	W =    -2.744 deg,	P =    30.268 deg,	R =  -167.022 deg
   GP2:
	UF : 1, UT : 1,
	J1=    90.000 deg,	J2=   -90.000 deg
};
P[599]{
   GP1:
	UF : 1, UT : 1,		CONFIG : 'N U T, 0, 0, 0',
	X =  2391.109  mm,	Y =   106.727  mm,	Z =   -21.577  mm,
	W =   -47.008 deg,	P =     6.653 deg,	R =   -83.994 deg
   GP2:
	UF : 1, UT : 1,
	J1=    83.000 deg,	J2=   -90.000 deg
};
P[600]{
   GP1:
	UF : 1, UT : 1,		CONFIG : 'N U T, 0, 0, 0',
	X =  2390.648  mm,	Y =   140.871  mm,	Z =   -20.910  mm,
	W =   -47.989 deg,	P =     7.881 deg,	R =   -87.078 deg
   GP2:
	UF : 1, UT : 1,
	J1=    83.000 deg,	J2=   -90.000 deg
};
P[601]{
   GP1:
	UF : 1, UT : 1,		CONFIG : 'N U T, 0, 0, 0',
	X =  2393.525  mm,	Y =   163.570  mm,	Z =   -20.785  mm,
	W =   -47.988 deg,	P =     7.880 deg,	R =  -106.126 deg
   GP2:
	UF : 1, UT : 1,
	J1=    83.000 deg,	J2=   -90.000 deg
};
P[602]{
   GP1:
	UF : 1, UT : 1,		CONFIG : 'N U T, 0, 0, 0',
	X =  2366.142  mm,	Y =   180.100  mm,	Z =    -9.199  mm,
	W =   -44.813 deg,	P =    -4.559 deg,	R =    -2.484 deg
   GP2:
	UF : 1, UT : 1,
	J1=    90.000 deg,	J2=   -90.000 deg
};
P[603]{
   GP1:
	UF : 1, UT : 1,		CONFIG : 'N U T, 0, 0, 0',
	X =  2505.035  mm,	Y =   180.287  mm,	Z =    -9.109  mm,
	W =   -44.818 deg,	P =    -4.562 deg,	R =    -2.490 deg
   GP2:
	UF : 1, UT : 1,
	J1=    90.000 deg,	J2=   -90.000 deg
};
P[604]{
   GP1:
	UF : 1, UT : 1,		CONFIG : 'N U T, 0, 0, 0',
	X =  2363.074  mm,	Y =    82.607  mm,	Z =    -8.621  mm,
	W =   -44.379 deg,	P =     8.160 deg,	R =    14.035 deg
   GP2:
	UF : 1, UT : 1,
	J1=    90.000 deg,	J2=   -90.000 deg
};
P[605]{
   GP1:
	UF : 1, UT : 1,		CONFIG : 'N U T, 0, 0, 0',
	X =  2414.311  mm,	Y =    81.629  mm,	Z =    -8.521  mm,
	W =   -44.393 deg,	P =     8.163 deg,	R =    14.043 deg
   GP2:
	UF : 1, UT : 1,
	J1=    90.000 deg,	J2=   -90.000 deg
};
P[606]{
   GP1:
	UF : 1, UT : 1,		CONFIG : 'N U T, 0, 0, 0',
	X =  2420.856  mm,	Y =    84.559  mm,	Z =    -6.348  mm,
	W =   -44.535 deg,	P =    -7.128 deg,	R =    33.228 deg
   GP2:
	UF : 1, UT : 1,
	J1=    90.000 deg,	J2=   -90.000 deg
};
P[607]{
   GP1:
	UF : 1, UT : 1,		CONFIG : 'N U T, 0, 0, 0',
	X =  2096.605  mm,	Y =  -181.583  mm,	Z =   897.867  mm,
	W =     -.064 deg,	P =    31.734 deg,	R =  -164.129 deg
   GP2:
	UF : 1, UT : 1,
	J1=    90.000 deg,	J2=   -90.000 deg
};
P[608]{
   GP1:
	UF : 1, UT : 1,		CONFIG : 'N U T, 0, 0, 0',
	X =  2114.149  mm,	Y =  -253.336  mm,	Z =   921.197  mm,
	W =     1.157 deg,	P =    35.359 deg,	R =   -90.786 deg
   GP2:
	UF : 1, UT : 1,
	J1=    90.000 deg,	J2=   -90.000 deg
};
P[609]{
   GP1:
	UF : 1, UT : 1,		CONFIG : 'N U T, 0, 0, 0',
	X =  2347.090  mm,	Y =    54.696  mm,	Z =   840.157  mm,
	W =    45.388 deg,	P =    17.262 deg,	R =    -1.525 deg
   GP2:
	UF : 1, UT : 1,
	J1=    90.000 deg,	J2=   -90.000 deg
};
P[610]{
   GP1:
	UF : 1, UT : 1,		CONFIG : 'N U T, 0, 0, 0',
	X =  2407.727  mm,	Y =    84.771  mm,	Z =   840.157  mm,
	W =    45.388 deg,	P =    17.262 deg,	R =    -1.525 deg
   GP2:
	UF : 1, UT : 1,
	J1=    90.000 deg,	J2=   -90.000 deg
};
P[611]{
   GP1:
	UF : 1, UT : 1,		CONFIG : 'N U T, 0, 0, 0',
	X =  2411.910  mm,	Y =    90.376  mm,	Z =   839.563  mm,
	W =     1.454 deg,	P =    40.369 deg,	R =    26.792 deg
   GP2:
	UF : 1, UT : 1,
	J1=    90.000 deg,	J2=   -90.000 deg
};
P[612]{
   GP1:
	UF : 1, UT : 1,		CONFIG : 'N U T, 0, 0, 0',
	X =  2400.458  mm,	Y =   114.292  mm,	Z =   839.623  mm,
	W =     1.448 deg,	P =    40.366 deg,	R =    26.776 deg
   GP2:
	UF : 1, UT : 1,
	J1=    90.000 deg,	J2=   -90.000 deg
};
P[613]{
   GP1:
	UF : 1, UT : 1,		CONFIG : 'N U T, 0, 0, 0',
	X =  2330.795  mm,	Y =    79.737  mm,	Z =   841.199  mm,
	W =   -50.335 deg,	P =   -10.786 deg,	R =    47.268 deg
   GP2:
	UF : 1, UT : 1,
	J1=    90.000 deg,	J2=   -90.000 deg
};
P[614]{
   GP1:
	UF : 1, UT : 1,		CONFIG : 'N U T, 0, 0, 0',
	X =  2394.366  mm,	Y =   112.525  mm,	Z =   840.958  mm,
	W =   -50.044 deg,	P =   -12.807 deg,	R =    45.682 deg
   GP2:
	UF : 1, UT : 1,
	J1=    90.000 deg,	J2=   -90.000 deg
};
P[615]{
   GP1:
	UF : 1, UT : 1,		CONFIG : 'N U T, 0, 0, 0',
	X =  2010.656  mm,	Y =   -98.489  mm,	Z =    -6.723  mm,
	W =    40.376 deg,	P =    23.931 deg,	R =    74.346 deg
   GP2:
	UF : 1, UT : 1,
	J1=    90.000 deg,	J2=  -100.000 deg
};
P[616]{
   GP1:
	UF : 1, UT : 1,		CONFIG : 'N U T, 0, 0, 0',
	X =  2009.129  mm,	Y =   124.302  mm,	Z =   -44.627  mm,
	W =    45.687 deg,	P =     4.511 deg,	R =    78.829 deg
   GP2:
	UF : 1, UT : 1,
	J1=    90.000 deg,	J2=  -100.000 deg
};
P[617]{
   GP1:
	UF : 1, UT : 1,		CONFIG : 'N U T, 0, 0, 0',
	X =  2230.271  mm,	Y =   -64.539  mm,	Z =    -1.822  mm,
	W =    44.892 deg,	P =    -3.427 deg,	R =     3.436 deg
   GP2:
	UF : 1, UT : 1,
	J1=    90.000 deg,	J2=   -90.000 deg
};
P[618]{
   GP1:
	UF : 1, UT : 1,		CONFIG : 'N U T, 0, 0, 0',
	X =  2628.655  mm,	Y =   126.905  mm,	Z =   907.127  mm,
	W =    31.997 deg,	P =    23.849 deg,	R =   -38.788 deg
   GP2:
	UF : 1, UT : 1,
	J1=    90.000 deg,	J2=   -90.000 deg
};
P[619]{
   GP1:
	UF : 1, UT : 1,		CONFIG : 'N U T, 0, 0, 0',
	X =   949.417  mm,	Y =    74.708  mm,	Z =  1003.698  mm,
	W =    14.657 deg,	P =    21.488 deg,	R =   -36.321 deg
   GP2:
	UF : 1, UT : 1,
	J1=    90.000 deg,	J2=   -90.000 deg
};
P[620]{
   GP1:
	UF : 1, UT : 1,		CONFIG : 'N U T, 0, 0, 0',
	X =   931.440  mm,	Y =   198.476  mm,	Z =   335.127  mm,
	W =   -34.527 deg,	P =    19.136 deg,	R =    25.896 deg
   GP2:
	UF : 1, UT : 1,
	J1=    90.000 deg,	J2=   -90.000 deg
};
P[621]{
   GP1:
	UF : 1, UT : 1,		CONFIG : 'N U T, 0, 0, 0',
	X =  1700.688  mm,	Y =   121.333  mm,	Z =   177.127  mm,
	W =   -48.737 deg,	P =     8.784 deg,	R =     7.978 deg
   GP2:
	UF : 1, UT : 1,
	J1=    90.000 deg,	J2=   -90.000 deg
};
P[622]{
   GP1:
	UF : 1, UT : 1,		CONFIG : 'N U T, 0, 0, 0',
	X =  2260.320  mm,	Y =   -63.687  mm,	Z =    -1.783  mm,
	W =    44.897 deg,	P =    -3.424 deg,	R =     3.430 deg
   GP2:
	UF : 1, UT : 1,
	J1=    90.000 deg,	J2=   -90.000 deg
};
P[623]{
   GP1:
	UF : 1, UT : 1,		CONFIG : 'N U T, 0, 0, 0',
	X =  2134.875  mm,	Y =   -62.293  mm,	Z =   -12.089  mm,
	W =    44.886 deg,	P =     3.630 deg,	R =    -4.912 deg
   GP2:
	UF : 1, UT : 1,
	J1=    90.000 deg,	J2=   -90.000 deg
};
P[624]{
   GP1:
	UF : 1, UT : 1,		CONFIG : 'N U T, 0, 0, 0',
	X =  2205.171  mm,	Y =   -64.816  mm,	Z =   -10.170  mm,
	W =    44.886 deg,	P =     3.630 deg,	R =    -4.912 deg
   GP2:
	UF : 1, UT : 1,
	J1=    90.000 deg,	J2=   -90.000 deg
};
P[625]{
   GP1:
	UF : 1, UT : 1,		CONFIG : 'N U T, 0, 0, 0',
	X =  2212.120  mm,	Y =   -62.897  mm,	Z =   -10.890  mm,
	W =    44.886 deg,	P =     3.630 deg,	R =   -11.550 deg
   GP2:
	UF : 1, UT : 1,
	J1=    90.000 deg,	J2=   -90.000 deg
};
P[626]{
   GP1:
	UF : 1, UT : 1,		CONFIG : 'N U T, 0, 0, 0',
	X =  1922.982  mm,	Y =    80.524  mm,	Z =   163.198  mm,
	W =   -51.903 deg,	P =     9.364 deg,	R =    21.482 deg
   GP2:
	UF : 1, UT : 1,
	J1=    90.000 deg,	J2=   -90.000 deg
};
P[627]{
   GP1:
	UF : 1, UT : 1,		CONFIG : 'N U T, 0, 0, 0',
	X =  2179.982  mm,	Y =    80.524  mm,	Z =   163.199  mm,
	W =   -51.227 deg,	P =   -13.564 deg,	R =     3.543 deg
   GP2:
	UF : 1, UT : 1,
	J1=    90.000 deg,	J2=   -90.000 deg
};
P[628]{
   GP1:
	UF : 1, UT : 1,		CONFIG : 'N U T, 0, 0, 0',
	X =  1984.534  mm,	Y =   -65.727  mm,	Z =   -17.955  mm,
	W =    44.885 deg,	P =     3.628 deg,	R =    -8.844 deg
   GP2:
	UF : 1, UT : 1,
	J1=    90.000 deg,	J2=   -90.000 deg
};
P[629]{
   GP1:
	UF : 1, UT : 1,		CONFIG : 'N U T, 0, 0, 0',
	X =  2097.268  mm,	Y =   -65.065  mm,	Z =   -17.473  mm,
	W =    44.885 deg,	P =     3.628 deg,	R =    -8.844 deg
   GP2:
	UF : 1, UT : 1,
	J1=    90.000 deg,	J2=   -90.000 deg
};
P[630]{
   GP1:
	UF : 1, UT : 1,		CONFIG : 'N U T, 0, 0, 0',
	X =  2179.963  mm,	Y =     8.530  mm,	Z =    59.476  mm,
	W =   -44.735 deg,	P =    -5.491 deg,	R =    -5.516 deg
   GP2:
	UF : 1, UT : 1,
	J1=    90.000 deg,	J2=   -90.000 deg
};
P[631]{
   GP1:
	UF : 1, UT : 1,		CONFIG : 'N U T, 0, 0, 0',
	X =  2112.828  mm,	Y =   -64.584  mm,	Z =   -16.753  mm,
	W =    41.205 deg,	P =   -19.972 deg,	R =    -8.013 deg
   GP2:
	UF : 1, UT : 1,
	J1=    90.000 deg,	J2=   -90.000 deg
};
P[632]{
   GP1:
	UF : 1, UT : 1,		CONFIG : 'N U T, 0, 0, 0',
	X =  2071.831  mm,	Y =  -111.826  mm,	Z =   -18.286  mm,
	W =   -37.503 deg,	P =      .971 deg,	R =    76.661 deg
   GP2:
	UF : 1, UT : 1,
	J1=    90.000 deg,	J2=   -90.000 deg
};
P[633]{
   GP1:
	UF : 1, UT : 1,		CONFIG : 'N U T, 0, 0, 0',
	X =  2101.801  mm,	Y =   -84.456  mm,	Z =   -18.286  mm,
	W =   -37.503 deg,	P =      .971 deg,	R =    85.242 deg
   GP2:
	UF : 1, UT : 1,
	J1=    90.000 deg,	J2=   -90.000 deg
};
P[634]{
   GP1:
	UF : 1, UT : 1,		CONFIG : 'N U T, 0, 0, 0',
	X =  2083.048  mm,	Y =     5.303  mm,	Z =    47.541  mm,
	W =   -44.735 deg,	P =    -5.491 deg,	R =    -5.516 deg
   GP2:
	UF : 1, UT : 1,
	J1=    90.000 deg,	J2=   -90.000 deg
};
P[635]{
   GP1:
	UF : 1, UT : 1,		CONFIG : 'N U T, 0, 0, 0',
	X =  2119.303  mm,	Y =   -69.097  mm,	Z =   -17.436  mm,
	W =   -37.503 deg,	P =      .971 deg,	R =   107.030 deg
   GP2:
	UF : 1, UT : 1,
	J1=    90.000 deg,	J2=   -90.000 deg
};
P[636]{
   GP1:
	UF : 1, UT : 1,		CONFIG : 'N U T, 0, 0, 1',
	X =  2129.923  mm,	Y =  -163.109  mm,	Z =   831.039  mm,
	W =     3.597 deg,	P =    39.858 deg,	R =  -158.843 deg
   GP2:
	UF : 1, UT : 1,
	J1=    90.000 deg,	J2=   -90.000 deg
};
P[637]{
   GP1:
	UF : 1, UT : 1,		CONFIG : 'N U T, 0, 0, 1',
	X =  2137.809  mm,	Y =  -186.248  mm,	Z =   831.044  mm,
	W =     2.770 deg,	P =    38.184 deg,	R =  -159.358 deg
   GP2:
	UF : 1, UT : 1,
	J1=    90.000 deg,	J2=   -90.000 deg
};
P[638]{
   GP1:
	UF : 1, UT : 1,		CONFIG : 'N U T, 0, 0, 0',
	X =  2065.479  mm,	Y =    84.939  mm,	Z =   110.355  mm,
	W =   -44.734 deg,	P =    -5.490 deg,	R =     4.917 deg
   GP2:
	UF : 1, UT : 1,
	J1=    90.000 deg,	J2=   -90.000 deg
};
P[639]{
   GP1:
	UF : 1, UT : 1,		CONFIG : 'N U T, 0, 0, 0',
	X =  1539.706  mm,	Y = -1470.455  mm,	Z =  1071.063  mm,
	W =   -42.856 deg,	P =   -15.293 deg,	R =    39.131 deg
   GP2:
	UF : 1, UT : 1,
	J1=   180.000 deg,	J2=  -125.000 deg
};
P[640]{
   GP1:
	UF : 1, UT : 1,		CONFIG : 'N U T, 0, 0, 0',
	X =  1166.553  mm,	Y = -1374.013  mm,	Z =  1522.225  mm,
	W =   -32.586 deg,	P =   -12.067 deg,	R =    17.529 deg
   GP2:
	UF : 1, UT : 1,
	J1=   180.000 deg,	J2=  -125.000 deg
};
P[641]{
   GP1:
	UF : 1, UT : 1,		CONFIG : 'N U T, 0, 0, 1',
	X =  1608.479  mm,	Y =   191.940  mm,	Z =    59.355  mm,
	W =    36.994 deg,	P =    27.707 deg,	R =  -122.588 deg
   GP2:
	UF : 1, UT : 1,
	J1=    90.000 deg,	J2=   -90.000 deg
};
P[642]{
   GP1:
	UF : 1, UT : 1,		CONFIG : 'N U T, 0, 0, 0',
	X =  2125.992  mm,	Y =  -204.644  mm,	Z =   830.285  mm,
	W =     7.244 deg,	P =    45.395 deg,	R =   112.852 deg
   GP2:
	UF : 1, UT : 1,
	J1=    90.000 deg,	J2=   -90.000 deg
};
P[643]{
   GP1:
	UF : 1, UT : 1,		CONFIG : 'N U T, 0, 0, 0',
	X =  2100.015  mm,	Y =  -196.039  mm,	Z =   828.573  mm,
	W =     5.322 deg,	P =    47.573 deg,	R =    22.949 deg
   GP2:
	UF : 1, UT : 1,
	J1=    90.000 deg,	J2=   -90.000 deg
};
P[644]{
   GP1:
	UF : 1, UT : 1,		CONFIG : 'N U T, 0, 0, 0',
	X =  2086.616  mm,	Y =  -152.754  mm,	Z =   828.880  mm,
	W =      .306 deg,	P =    46.787 deg,	R =    19.130 deg
   GP2:
	UF : 1, UT : 1,
	J1=    90.000 deg,	J2=   -90.000 deg
};
P[645]{
   GP1:
	UF : 1, UT : 1,		CONFIG : 'N U T, 0, 0, 0',
	X =  1450.805  mm,	Y =    56.341  mm,	Z =   141.822  mm,
	W =    36.993 deg,	P =    27.706 deg,	R =  -154.189 deg
   GP2:
	UF : 1, UT : 1,
	J1=    90.000 deg,	J2=   -90.000 deg
};
P[646]{
   GP1:
	UF : 1, UT : 1,		CONFIG : 'N U T, 0, 0, 0',
	X =  1476.806  mm,	Y =   169.341  mm,	Z =   386.823  mm,
	W =    23.939 deg,	P =    39.314 deg,	R =  -177.488 deg
   GP2:
	UF : 1, UT : 1,
	J1=    80.000 deg,	J2=   -90.000 deg
};
P[647]{
   GP1:
	UF : 1, UT : 1,		CONFIG : 'N U T, 0, 0, 0',
	X =  2034.807  mm,	Y =   169.341  mm,	Z =   186.823  mm,
	W =    23.939 deg,	P =    39.314 deg,	R =  -177.488 deg
   GP2:
	UF : 1, UT : 1,
	J1=    80.000 deg,	J2=   -90.000 deg
};
P[648]{
   GP1:
	UF : 1, UT : 1,		CONFIG : 'N U T, 0, 0, -1',
	X =  2034.807  mm,	Y =     1.341  mm,	Z =   115.823  mm,
	W =    34.881 deg,	P =    30.459 deg,	R =  -142.693 deg
   GP2:
	UF : 1, UT : 1,
	J1=    80.000 deg,	J2=   -90.000 deg
};
P[649]{
   GP1:
	UF : 1, UT : 1,		CONFIG : 'N U T, 0, 0, 0',
	X =  2100.504  mm,	Y =  -134.531  mm,	Z =   832.401  mm,
	W =    -1.751 deg,	P =    45.025 deg,	R =   -76.985 deg
   GP2:
	UF : 1, UT : 1,
	J1=    90.000 deg,	J2=   -90.000 deg
};
P[650]{
   GP1:
	UF : 1, UT : 1,		CONFIG : 'N U T, 0, 0, 0',
	X =  2125.547  mm,	Y =  -142.237  mm,	Z =   829.698  mm,
	W =      .707 deg,	P =    41.168 deg,	R =  -163.588 deg
   GP2:
	UF : 1, UT : 1,
	J1=    90.000 deg,	J2=   -90.000 deg
};
P[651]{
   GP1:
	UF : 1, UT : 1,		CONFIG : 'N U T, 0, 0, 0',
	X =  2131.397  mm,	Y =  -162.602  mm,	Z =   829.829  mm,
	W =      .078 deg,	P =    40.942 deg,	R =  -164.204 deg
   GP2:
	UF : 1, UT : 1,
	J1=    90.000 deg,	J2=   -90.000 deg
};
P[652]{
   GP1:
	UF : 1, UT : 1,		CONFIG : 'N U T, 0, 0, 0',
	X =  2108.961  mm,	Y =  -235.302  mm,	Z =   830.555  mm,
	W =     -.443 deg,	P =    39.555 deg,	R =   -90.699 deg
   GP2:
	UF : 1, UT : 1,
	J1=    90.000 deg,	J2=   -90.000 deg
};
P[653]{
   GP1:
	UF : 1, UT : 1,		CONFIG : 'N U T, 0, 0, 0',
	X =  2201.336  mm,	Y =  -235.279  mm,	Z =   830.597  mm,
	W =     -.447 deg,	P =    39.555 deg,	R =   -90.703 deg
   GP2:
	UF : 1, UT : 1,
	J1=    90.000 deg,	J2=   -90.000 deg
};
P[654]{
   GP1:
	UF : 1, UT : 1,		CONFIG : 'N U T, 0, 0, 0',
	X =  2214.980  mm,	Y =  -233.048  mm,	Z =   831.869  mm,
	W =     -.447 deg,	P =    39.555 deg,	R =   -57.817 deg
   GP2:
	UF : 1, UT : 1,
	J1=    90.000 deg,	J2=   -90.000 deg
};
P[655]{
   GP1:
	UF : 1, UT : 1,		CONFIG : 'N U T, 0, 0, 0',
	X =  2222.918  mm,	Y =  -224.326  mm,	Z =   830.599  mm,
	W =     -.447 deg,	P =    39.555 deg,	R =   -44.058 deg
   GP2:
	UF : 1, UT : 1,
	J1=    90.000 deg,	J2=   -90.000 deg
};
P[656]{
   GP1:
	UF : 1, UT : 1,		CONFIG : 'N U T, 0, 0, 0',
	X =  2394.178  mm,	Y =   -28.001  mm,	Z =   831.741  mm,
	W =     -.034 deg,	P =    41.997 deg,	R =   -43.180 deg
   GP2:
	UF : 1, UT : 1,
	J1=    90.000 deg,	J2=   -90.000 deg
};
P[657]{
   GP1:
	UF : 1, UT : 1,		CONFIG : 'N U T, 0, 0, 0',
	X =  2450.792  mm,	Y =    35.777  mm,	Z =   832.312  mm,
	W =      .115 deg,	P =    42.764 deg,	R =   -49.054 deg
   GP2:
	UF : 1, UT : 1,
	J1=    90.000 deg,	J2=   -90.000 deg
};
P[658]{
   GP1:
	UF : 1, UT : 1,		CONFIG : 'N U T, 0, 0, 0',
	X =  2457.628  mm,	Y =    40.947  mm,	Z =   832.314  mm,
	W =      .115 deg,	P =    42.764 deg,	R =   -56.123 deg
   GP2:
	UF : 1, UT : 1,
	J1=    90.000 deg,	J2=   -90.000 deg
};
P[659]{
   GP1:
	UF : 1, UT : 1,		CONFIG : 'N U T, 0, 0, 0',
	X =  2521.514  mm,	Y =    87.672  mm,	Z =   832.133  mm,
	W =    11.971 deg,	P =    40.663 deg,	R =   -38.122 deg
   GP2:
	UF : 1, UT : 1,
	J1=    90.000 deg,	J2=   -90.000 deg
};
P[660]{
   GP1:
	UF : 1, UT : 1,		CONFIG : 'N U T, 0, 0, 0',
	X =  2650.676  mm,	Y =   184.582  mm,	Z =   832.304  mm,
	W =    27.597 deg,	P =    31.501 deg,	R =   -10.869 deg
   GP2:
	UF : 1, UT : 1,
	J1=    90.000 deg,	J2=   -90.000 deg
};
P[661]{
   GP1:
	UF : 1, UT : 1,		CONFIG : 'N U T, 0, 0, 0',
	X =  1959.340  mm,	Y =   -50.107  mm,	Z =    51.552  mm,
	W =   -51.898 deg,	P =     9.370 deg,	R =    14.305 deg
   GP2:
	UF : 1, UT : 1,
	J1=    90.000 deg,	J2=   -90.000 deg
};
P[662]{
   GP1:
	UF : 1, UT : 1,		CONFIG : 'N U T, 0, 0, 0',
	X =  1948.268  mm,	Y =   -49.653  mm,	Z =    51.537  mm,
	W =   -51.894 deg,	P =     9.366 deg,	R =     5.846 deg
   GP2:
	UF : 1, UT : 1,
	J1=    90.000 deg,	J2=   -90.000 deg
};
P[663]{
   GP1:
	UF : 1, UT : 1,		CONFIG : 'N U T, 0, 0, 0',
	X =  1696.243  mm,	Y =   -50.530  mm,	Z =    52.257  mm,
	W =   -51.894 deg,	P =     9.366 deg,	R =     5.846 deg
   GP2:
	UF : 1, UT : 1,
	J1=    90.000 deg,	J2=   -90.000 deg
};
P[664]{
   GP1:
	UF : 1, UT : 1,		CONFIG : 'N U T, 0, 0, 0',
	X =  1670.714  mm,	Y =   -48.833  mm,	Z =    54.913  mm,
	W =   -51.894 deg,	P =     9.366 deg,	R =   -32.596 deg
   GP2:
	UF : 1, UT : 1,
	J1=    90.000 deg,	J2=   -90.000 deg
};
P[665]{
   GP1:
	UF : 1, UT : 1,		CONFIG : 'N U T, 0, 0, 0',
	X =  2224.519  mm,	Y =   -44.534  mm,	Z =    -1.819  mm,
	W =   -45.065 deg,	P =    -5.943 deg,	R =    -3.250 deg
   GP2:
	UF : 1, UT : 1,
	J1=    90.000 deg,	J2=   -90.000 deg
};
P[666]{
   GP1:
	UF : 1, UT : 1,		CONFIG : 'N U T, 0, 0, 0',
	X =  2262.967  mm,	Y =   -46.459  mm,	Z =    -2.708  mm,
	W =   -45.063 deg,	P =    -5.948 deg,	R =    -3.255 deg
   GP2:
	UF : 1, UT : 1,
	J1=    90.000 deg,	J2=   -90.000 deg
};
P[667]{
   GP1:
	UF : 1, UT : 1,		CONFIG : 'N U T, 0, 0, 0',
	X =  2141.111  mm,	Y =   -46.149  mm,	Z =    -9.294  mm,
	W =   -44.730 deg,	P =    -5.491 deg,	R =    -5.523 deg
   GP2:
	UF : 1, UT : 1,
	J1=    90.000 deg,	J2=   -90.000 deg
};
P[668]{
   GP1:
	UF : 1, UT : 1,		CONFIG : 'N U T, 0, 0, 0',
	X =  2205.054  mm,	Y =   -46.149  mm,	Z =    -9.294  mm,
	W =   -44.730 deg,	P =    -5.491 deg,	R =    -5.523 deg
   GP2:
	UF : 1, UT : 1,
	J1=    90.000 deg,	J2=   -90.000 deg
};
P[669]{
   GP1:
	UF : 1, UT : 1,		CONFIG : 'N U T, 0, 0, 0',
	X =  2212.135  mm,	Y =   -45.578  mm,	Z =    -9.294  mm,
	W =   -44.730 deg,	P =    -5.491 deg,	R =    10.504 deg
   GP2:
	UF : 1, UT : 1,
	J1=    90.000 deg,	J2=   -90.000 deg
};
P[670]{
   GP1:
	UF : 1, UT : 1,		CONFIG : 'N U T, 0, 0, 0',
	X =  2492.536  mm,	Y =   739.403  mm,	Z =    25.184  mm,
	W =   -42.166 deg,	P =     5.515 deg,	R =   107.587 deg
   GP2:
	UF : 1, UT : 1,
	J1=    80.000 deg,	J2=   -90.000 deg
};
P[671]{
   GP1:
	UF : 1, UT : 1,		CONFIG : 'N U T, 0, 0, 0',
	X =  2492.536  mm,	Y =   809.403  mm,	Z =    25.184  mm,
	W =   -38.452 deg,	P =    19.595 deg,	R =   124.425 deg
   GP2:
	UF : 1, UT : 1,
	J1=    80.000 deg,	J2=   -90.000 deg
};
P[672]{
   GP1:
	UF : 1, UT : 1,		CONFIG : 'N U T, 0, 0, 0',
	X =  2115.729  mm,	Y =   -45.526  mm,	Z =   -17.679  mm,
	W =   -44.735 deg,	P =    -5.490 deg,	R =    -5.517 deg
   GP2:
	UF : 1, UT : 1,
	J1=    90.000 deg,	J2=   -90.000 deg
};
P[673]{
   GP1:
	UF : 1, UT : 1,		CONFIG : 'N U T, 0, 0, 0',
	X =  2032.308  mm,	Y =   -46.092  mm,	Z =   -17.679  mm,
	W =   -44.735 deg,	P =    -5.490 deg,	R =    -5.517 deg
   GP2:
	UF : 1, UT : 1,
	J1=    90.000 deg,	J2=   -90.000 deg
};
P[674]{
   GP1:
	UF : 1, UT : 1,		CONFIG : 'N U T, 0, 0, 0',
	X =  2010.263  mm,	Y =   -47.292  mm,	Z =   -17.680  mm,
	W =   -44.735 deg,	P =    -5.490 deg,	R =   -41.540 deg
   GP2:
	UF : 1, UT : 1,
	J1=    90.000 deg,	J2=   -90.000 deg
};
P[675]{
   GP1:
	UF : 1, UT : 1,		CONFIG : 'N U T, 0, 0, 0',
	X =  1652.956  mm,	Y =   215.868  mm,	Z =   -13.936  mm,
	W =    34.857 deg,	P =    26.466 deg,	R =  -126.842 deg
   GP2:
	UF : 1, UT : 1,
	J1=    90.000 deg,	J2=   -90.000 deg
};
P[676]{
   GP1:
	UF : 1, UT : 1,		CONFIG : 'N U T, 0, 0, 1',
	X =  1654.227  mm,	Y =    -6.870  mm,	Z =   -18.681  mm,
	W =    36.965 deg,	P =    27.690 deg,	R =  -122.601 deg
   GP2:
	UF : 1, UT : 1,
	J1=    90.000 deg,	J2=   -90.000 deg
};
P[677]{
   GP1:
	UF : 1, UT : 1,		CONFIG : 'N U T, 0, 0, 0',
	X =  1654.396  mm,	Y =   -25.585  mm,	Z =   -18.765  mm,
	W =    37.080 deg,	P =    27.790 deg,	R =  -137.819 deg
   GP2:
	UF : 1, UT : 1,
	J1=    90.000 deg,	J2=   -90.000 deg
};
P[678]{
   GP1:
	UF : 1, UT : 1,		CONFIG : 'N U T, 0, 0, 0',
	X =  2063.360  mm,	Y =   -46.552  mm,	Z =    14.408  mm,
	W =    27.118 deg,	P =    24.034 deg,	R =  -162.974 deg
   GP2:
	UF : 1, UT : 1,
	J1=    80.000 deg,	J2=   -90.000 deg
};
P[679]{
   GP1:
	UF : 1, UT : 1,		CONFIG : 'N U T, 0, 0, 0',
	X =  2521.799  mm,	Y =   685.855  mm,	Z =   110.598  mm,
	W =   -11.653 deg,	P =   -32.812 deg,	R =    68.201 deg
   GP2:
	UF : 1, UT : 1,
	J1=    80.000 deg,	J2=   -90.000 deg
};
P[680]{
   GP1:
	UF : 1, UT : 1,		CONFIG : 'N U T, 0, 0, 0',
	X =  2352.111  mm,	Y =   297.878  mm,	Z =   188.758  mm,
	W =   -43.260 deg,	P =    61.542 deg,	R =   123.185 deg
   GP2:
	UF : 1, UT : 1,
	J1=    80.000 deg,	J2=   -90.000 deg
};
P[681]{
   GP1:
	UF : 1, UT : 1,		CONFIG : 'N U T, 0, 0, 0',
	X =  1368.100  mm,	Y =   306.117  mm,	Z =   479.720  mm,
	W =   -19.454 deg,	P =    45.370 deg,	R =   135.446 deg
   GP2:
	UF : 1, UT : 1,
	J1=    80.000 deg,	J2=   -90.000 deg
};
P[682]{
   GP1:
	UF : 1, UT : 1,		CONFIG : 'N U T, 0, 0, 0',
	X =   586.370  mm,	Y =  -785.188  mm,	Z =  2292.509  mm,
	W =   -20.678 deg,	P =   -36.657 deg,	R =     1.573 deg
   GP2:
	UF : 1, UT : 1,
	J1=   180.000 deg,	J2=  -150.000 deg
};
P[683]{
   GP1:
	UF : 1, UT : 1,		CONFIG : 'N U T, 0, 0, 0',
	X =   642.423  mm,	Y = -1094.246  mm,	Z =  1725.795  mm,
	W =     2.647 deg,	P =   -31.291 deg,	R =   -11.601 deg
   GP2:
	UF : 1, UT : 1,
	J1=   180.000 deg,	J2=  -150.000 deg
};
P[684]{
   GP1:
	UF : 1, UT : 1,		CONFIG : 'N U T, 0, 0, 0',
	X =   799.244  mm,	Y = -1202.971  mm,	Z =  1035.322  mm,
	W =    24.190 deg,	P =   -39.178 deg,	R =    -6.255 deg
   GP2:
	UF : 1, UT : 1,
	J1=   180.000 deg,	J2=  -150.000 deg
};
P[685]{
   GP1:
	UF : 1, UT : 1,		CONFIG : 'N U T, 0, 0, 0',
	X =   954.244  mm,	Y = -1102.971  mm,	Z =   861.322  mm,
	W =    24.190 deg,	P =   -39.178 deg,	R =    -6.255 deg
   GP2:
	UF : 1, UT : 1,
	J1=   180.000 deg,	J2=  -150.000 deg
};
P[686]{
   GP1:
	UF : 1, UT : 1,		CONFIG : 'N U T, 0, 0, 1',
	X =  2070.201  mm,	Y =    -5.697  mm,	Z =    13.112  mm,
	W =    26.540 deg,	P =    23.909 deg,	R =  -139.397 deg
   GP2:
	UF : 0, UT : 1,
	J1=    80.000 deg,	J2=   -90.000 deg
};
P[687]{
   GP1:
	UF : 1, UT : 1,		CONFIG : 'N U T, 0, 0, 0',
	X =  2069.499  mm,	Y =    -1.522  mm,	Z =    13.452  mm,
	W =    26.543 deg,	P =    23.908 deg,	R =  -163.851 deg
   GP2:
	UF : 1, UT : 1,
	J1=    80.000 deg,	J2=   -90.000 deg
};
P[688]{
   GP1:
	UF : 1, UT : 1,		CONFIG : 'N U T, 0, 0, 0',
	X =   955.526  mm,	Y = -1174.727  mm,	Z =   902.888  mm,
	W =    27.863 deg,	P =   -46.318 deg,	R =   -16.260 deg
   GP2:
	UF : 1, UT : 1,
	J1=   180.000 deg,	J2=  -150.000 deg
};
P[689]{
   GP1:
	UF : 1, UT : 1,		CONFIG : 'N U T, 0, 0, 0',
	X =   571.093  mm,	Y = -1097.630  mm,	Z =  1035.072  mm,
	W =    42.871 deg,	P =   -15.240 deg,	R =   -45.029 deg
   GP2:
	UF : 1, UT : 1,
	J1=   180.000 deg,	J2=  -150.000 deg
};
P[690]{
   GP1:
	UF : 1, UT : 1,		CONFIG : 'N U T, 0, 0, 0',
	X =   749.093  mm,	Y =  -654.630  mm,	Z =   835.073  mm,
	W =    44.064 deg,	P =   -10.243 deg,	R =   -50.428 deg
   GP2:
	UF : 1, UT : 1,
	J1=   180.000 deg,	J2=  -150.000 deg
};
P[691]{
   GP1:
	UF : 1, UT : 1,		CONFIG : 'N U T, 0, 0, 0',
	X =  2079.957  mm,	Y =    14.618  mm,	Z =    14.062  mm,
	W =    17.949 deg,	P =    33.023 deg,	R =   153.341 deg
   GP2:
	UF : 1, UT : 1,
	J1=    80.000 deg,	J2=   -90.000 deg
};
P[692]{
   GP1:
	UF : 1, UT : 1,		CONFIG : 'N U T, 0, 0, 0',
	X =  2257.638  mm,	Y =   188.605  mm,	Z =   -17.721  mm,
	W =      .048 deg,	P =    36.127 deg,	R =   125.240 deg
   GP2:
	UF : 0, UT : 1,
	J1=    80.000 deg,	J2=   -90.000 deg
};
P[693]{
   GP1:
	UF : 1, UT : 1,		CONFIG : 'N U T, 0, 0, 0',
	X =  2269.957  mm,	Y =   197.647  mm,	Z =   -19.138  mm,
	W =     3.307 deg,	P =    33.871 deg,	R =   124.431 deg
   GP2:
	UF : 0, UT : 1,
	J1=    80.000 deg,	J2=   -90.000 deg
};
P[694]{
   GP1:
	UF : 1, UT : 1,		CONFIG : 'N U T, 0, 0, 0',
	X =   962.545  mm,	Y = -1093.036  mm,	Z =   867.966  mm,
	W =    44.863 deg,	P =     3.974 deg,	R =   -63.984 deg
   GP2:
	UF : 1, UT : 1,
	J1=   180.000 deg,	J2=  -150.000 deg
};
P[695]{
   GP1:
	UF : 1, UT : 1,		CONFIG : 'N U T, 0, 0, 0',
	X =   592.698  mm,	Y =  -634.536  mm,	Z =   863.966  mm,
	W =    36.388 deg,	P =   -28.554 deg,	R =   -27.033 deg
   GP2:
	UF : 1, UT : 1,
	J1=   180.000 deg,	J2=  -150.000 deg
};
P[696]{
   GP1:
	UF : 1, UT : 1,		CONFIG : 'N U T, 0, 0, 0',
	X =  2281.172  mm,	Y =   204.541  mm,	Z =   -20.943  mm,
	W =     6.003 deg,	P =    35.927 deg,	R =   123.386 deg
   GP2:
	UF : 0, UT : 1,
	J1=    80.000 deg,	J2=   -90.000 deg
};
P[697]{
   GP1:
	UF : 1, UT : 1,		CONFIG : 'N U T, 0, 0, 0',
	X =  2386.760  mm,	Y =   271.261  mm,	Z =   -38.436  mm,
	W =     8.791 deg,	P =    37.202 deg,	R =   129.076 deg
   GP2:
	UF : 0, UT : 1,
	J1=    80.000 deg,	J2=   -90.000 deg
};
P[698]{
   GP1:
	UF : 1, UT : 1,		CONFIG : 'N U T, 0, 0, 0',
	X =   545.804  mm,	Y =  -597.246  mm,	Z =   979.702  mm,
	W =    15.937 deg,	P =   -42.493 deg,	R =     6.853 deg
   GP2:
	UF : 1, UT : 1,
	J1=   180.000 deg,	J2=  -150.000 deg
};
P[699]{
   GP1:
	UF : 1, UT : 1,		CONFIG : 'N U T, 0, 0, 0',
	X =   366.532  mm,	Y =  -833.172  mm,	Z =  1480.397  mm,
	W =    13.558 deg,	P =     8.679 deg,	R =   -55.514 deg
   GP2:
	UF : 1, UT : 1,
	J1=   180.000 deg,	J2=  -150.000 deg
};
P[700]{
   GP1:
	UF : 1, UT : 1,		CONFIG : 'N U T, 0, 0, 0',
	X =  1532.562  mm,	Y = -1156.369  mm,	Z =  1523.814  mm,
	W =   -53.323 deg,	P =    -7.912 deg,	R =   -20.862 deg
   GP2:
	UF : 0, UT : 1,
	J1=   180.000 deg,	J2=   -90.000 deg
};
P[701]{
   GP1:
	UF : 1, UT : 1,		CONFIG : 'N U T, 0, 0, 0',
	X =  1863.519  mm,	Y = -1304.565  mm,	Z =  1265.460  mm,
	W =   -45.547 deg,	P =    -6.107 deg,	R =    -5.943 deg
   GP2:
	UF : 0, UT : 1,
	J1=   180.000 deg,	J2=   -90.000 deg
};
P[702]{
   GP1:
	UF : 1, UT : 1,		CONFIG : 'N U T, 0, 0, 0',
	X =  1929.519  mm,	Y = -1405.565  mm,	Z =  1058.460  mm,
	W =   -42.701 deg,	P =    18.644 deg,	R =    19.122 deg
   GP2:
	UF : 0, UT : 1,
	J1=   180.000 deg,	J2=   -90.000 deg
};
P[703]{
   GP1:
	UF : 1, UT : 1,		CONFIG : 'N U T, 0, 0, 0',
	X =  2402.059  mm,	Y =   281.172  mm,	Z =   -42.884  mm,
	W =    -2.502 deg,	P =    34.195 deg,	R =   123.652 deg
   GP2:
	UF : 0, UT : 1,
	J1=    80.000 deg,	J2=   -90.000 deg
};
P[704]{
   GP1:
	UF : 1, UT : 1,		CONFIG : 'N U T, 0, 0, 0',
	X =  2416.336  mm,	Y =   299.753  mm,	Z =   -44.208  mm,
	W =      .578 deg,	P =    31.078 deg,	R =   135.858 deg
   GP2:
	UF : 0, UT : 1,
	J1=    80.000 deg,	J2=   -90.000 deg
};
P[705]{
   GP1:
	UF : 1, UT : 1,		CONFIG : 'N U T, 0, 0, 0',
	X =  2499.975  mm,	Y =   418.494  mm,	Z =   -59.863  mm,
	W =   -18.687 deg,	P =    29.860 deg,	R =   100.231 deg
   GP2:
	UF : 0, UT : 1,
	J1=    80.000 deg,	J2=   -90.000 deg
};
P[706]{
   GP1:
	UF : 1, UT : 1,		CONFIG : 'N U T, 0, 0, 0',
	X =  2522.749  mm,	Y =   437.814  mm,	Z =   -61.500  mm,
	W =   -18.823 deg,	P =    32.557 deg,	R =    79.853 deg
   GP2:
	UF : 0, UT : 1,
	J1=    80.000 deg,	J2=   -90.000 deg
};
P[707]{
   GP1:
	UF : 1, UT : 1,		CONFIG : 'N U T, 0, 0, 0',
	X =  2555.836  mm,	Y =   446.395  mm,	Z =   -68.337  mm,
	W =   -16.509 deg,	P =    33.836 deg,	R =    74.966 deg
   GP2:
	UF : 0, UT : 1,
	J1=    80.000 deg,	J2=   -90.000 deg
};
P[708]{
   GP1:
	UF : 1, UT : 1,		CONFIG : 'N U T, 0, 0, 0',
	X =  2039.010  mm,	Y = -1381.508  mm,	Z =  1071.568  mm,
	W =   -44.862 deg,	P =     3.961 deg,	R =   -20.537 deg
   GP2:
	UF : 0, UT : 1,
	J1=   180.000 deg,	J2=   -90.000 deg
};
P[709]{
   GP1:
	UF : 1, UT : 1,		CONFIG : 'N U T, 0, 0, 0',
	X =  2568.335  mm,	Y =   451.071  mm,	Z =   -68.337  mm,
	W =   -16.509 deg,	P =    33.836 deg,	R =    74.966 deg
   GP2:
	UF : 0, UT : 1,
	J1=    80.000 deg,	J2=   -90.000 deg
};
P[710]{
   GP1:
	UF : 1, UT : 1,		CONFIG : 'N U T, 0, 0, 0',
	X =  1822.564  mm,	Y = -1057.861  mm,	Z =  1463.123  mm,
	W =   -36.308 deg,	P =    -6.286 deg,	R =   -23.397 deg
   GP2:
	UF : 1, UT : 1,
	J1=   180.000 deg,	J2=   -90.000 deg
};
P[711]{
   GP1:
	UF : 1, UT : 1,		CONFIG : 'N U T, 0, 0, 0',
	X =  1392.804  mm,	Y =   640.782  mm,	Z =  1670.105  mm,
	W =    37.735 deg,	P =   -20.539 deg,	R =     -.894 deg
   GP2:
	UF : 0, UT : 1,
	J1=   180.000 deg,	J2=    90.000 deg
};
P[712]{
   GP1:
	UF : 1, UT : 1,		CONFIG : 'N U T, 0, 0, 0',
	X =  1849.519  mm,	Y =  1220.906  mm,	Z =  1351.461  mm,
	W =    44.958 deg,	P =    -2.212 deg,	R =     2.229 deg
   GP2:
	UF : 0, UT : 1,
	J1=   180.000 deg,	J2=    90.000 deg
};
P[713]{
   GP1:
	UF : 1, UT : 1,		CONFIG : 'N U T, 0, 0, 0',
	X =  1880.451  mm,	Y =  1275.016  mm,	Z =  1238.303  mm,
	W =    44.592 deg,	P =     6.805 deg,	R =    -6.838 deg
   GP2:
	UF : 1, UT : 1,
	J1=   180.000 deg,	J2=    90.000 deg
};
P[714]{
   GP1:
	UF : 1, UT : 1,		CONFIG : 'N U T, 0, 0, 0',
	X =  1926.400  mm,	Y =  1355.399  mm,	Z =  1070.204  mm,
	W =    41.277 deg,	P =    19.800 deg,	R =   -21.086 deg
   GP2:
	UF : 0, UT : 1,
	J1=   180.000 deg,	J2=    90.000 deg
};
P[715]{
   GP1:
	UF : 1, UT : 1,		CONFIG : 'N U T, 0, 0, 0',
	X =  2604.215  mm,	Y =   477.246  mm,	Z =   -76.736  mm,
	W =   -17.687 deg,	P =    33.474 deg,	R =   110.394 deg
   GP2:
	UF : 0, UT : 1,
	J1=    80.000 deg,	J2=   -90.000 deg
};
P[716]{
   GP1:
	UF : 1, UT : 1,		CONFIG : 'N U T, 0, 0, 0',
	X =  2618.697  mm,	Y =   518.470  mm,	Z =   -81.888  mm,
	W =   -28.179 deg,	P =    11.270 deg,	R =   110.042 deg
   GP2:
	UF : 0, UT : 1,
	J1=    80.000 deg,	J2=   -90.000 deg
};
P[717]{
   GP1:
	UF : 1, UT : 1,		CONFIG : 'N U T, 0, 0, 0',
	X =  2619.516  mm,	Y =   709.528  mm,	Z =   -82.638  mm,
	W =   -28.920 deg,	P =    12.962 deg,	R =   109.018 deg
   GP2:
	UF : 0, UT : 1,
	J1=    80.000 deg,	J2=   -90.000 deg
};
P[718]{
   GP1:
	UF : 1, UT : 1,		CONFIG : 'N U T, 0, 0, 0',
	X =  2621.157  mm,	Y =   717.292  mm,	Z =   -84.163  mm,
	W =   -28.920 deg,	P =    12.962 deg,	R =    86.656 deg
   GP2:
	UF : 0, UT : 1,
	J1=    80.000 deg,	J2=   -90.000 deg
};
P[719]{
   GP1:
	UF : 1, UT : 1,		CONFIG : 'N U T, 0, 0, 0',
	X =  2623.715  mm,	Y =   724.341  mm,	Z =   -84.162  mm,
	W =   -28.920 deg,	P =    12.962 deg,	R =    81.288 deg
   GP2:
	UF : 0, UT : 1,
	J1=    80.000 deg,	J2=   -90.000 deg
};
P[720]{
   GP1:
	UF : 1, UT : 1,		CONFIG : 'N U T, 0, 0, 0',
	X =  1993.007  mm,	Y =  1431.170  mm,	Z =  1068.677  mm,
	W =    44.305 deg,	P =     8.850 deg,	R =     3.803 deg
   GP2:
	UF : 1, UT : 1,
	J1=   180.000 deg,	J2=    90.000 deg
};
P[721]{
   GP1:
	UF : 1, UT : 1,		CONFIG : 'N U T, 0, 0, 0',
	X =  1840.948  mm,	Y =  1174.835  mm,	Z =  1330.032  mm,
	W =    44.958 deg,	P =    -2.212 deg,	R =     2.229 deg
   GP2:
	UF : 0, UT : 1,
	J1=   180.000 deg,	J2=    90.000 deg
};
P[722]{
   GP1:
	UF : 1, UT : 1,		CONFIG : 'N U T, 0, 0, 0',
	X =  2631.075  mm,	Y =   754.747  mm,	Z =   -85.027  mm,
	W =   -29.833 deg,	P =     9.276 deg,	R =    88.853 deg
   GP2:
	UF : 0, UT : 1,
	J1=    80.000 deg,	J2=   -90.000 deg
};
P[723]{
   GP1:
	UF : 1, UT : 1,		CONFIG : 'N U T, 0, 0, 0',
	X =  2630.091  mm,	Y =   766.127  mm,	Z =   -86.552  mm,
	W =   -33.769 deg,	P =      .741 deg,	R =   112.878 deg
   GP2:
	UF : 0, UT : 1,
	J1=    80.000 deg,	J2=   -90.000 deg
};
P[731]{
   GP1:
	UF : 1, UT : 1,		CONFIG : 'N U T, 0, 0, 0',
	X =  1053.046  mm,	Y = -1056.747  mm,	Z =   769.543  mm,
	W =    24.542 deg,	P =   -38.984 deg,	R =    -6.156 deg
   GP2:
	UF : 1, UT : 1,
	J1=   180.000 deg,	J2=  -150.000 deg
};
P[732]{
   GP1:
	UF : 1, UT : 1,		CONFIG : 'F U T, 0, 0, 0',
	X =   804.374  mm,	Y =   981.069  mm,	Z =  1117.927  mm,
	W =    50.730 deg,	P =      .639 deg,	R =   -51.736 deg
   GP2:
	UF : 1, UT : 1,
	J1=   180.000 deg,	J2=   150.000 deg
};
P[733]{
   GP1:
	UF : 1, UT : 1,		CONFIG : 'F U T, 0, 0, 0',
	X =  1064.016  mm,	Y =   999.283  mm,	Z =  1072.926  mm,
	W =    50.730 deg,	P =      .639 deg,	R =   -51.736 deg
   GP2:
	UF : 1, UT : 1,
	J1=   180.000 deg,	J2=   150.000 deg
};
P[734]{
   GP1:
	UF : 1, UT : 1,		CONFIG : 'N U T, 0, 0, 0',
	X =  1094.890  mm,	Y = -1127.769  mm,	Z =   768.463  mm,
	W =    24.536 deg,	P =   -38.987 deg,	R =    -6.145 deg
   GP2:
	UF : 1, UT : 1,
	J1=   180.000 deg,	J2=  -150.000 deg
};
P[735]{
   GP1:
	UF : 1, UT : 1,		CONFIG : 'N U T, 0, 0, 0',
	X =   776.756  mm,	Y =  -578.766  mm,	Z =   774.376  mm,
	W =    32.518 deg,	P =   -31.098 deg,	R =   -20.599 deg
   GP2:
	UF : 1, UT : 1,
	J1=   180.000 deg,	J2=  -150.000 deg
};
P[736]{
   GP1:
	UF : 1, UT : 1,		CONFIG : 'N U T, 0, 0, 0',
	X =   923.650  mm,	Y =  -831.496  mm,	Z =   772.822  mm,
	W =    41.898 deg,	P =   -14.128 deg,	R =   -49.385 deg
   GP2:
	UF : 1, UT : 1,
	J1=   180.000 deg,	J2=  -150.000 deg
};
P[737]{
   GP1:
	UF : 1, UT : 1,		CONFIG : 'N U T, 0, 0, 0',
	X =  1037.419  mm,	Y = -1025.988  mm,	Z =   770.961  mm,
	W =    43.034 deg,	P =    -8.862 deg,	R =   -55.276 deg
   GP2:
	UF : 1, UT : 1,
	J1=   180.000 deg,	J2=  -150.000 deg
};
P[738]{
   GP1:
	UF : 1, UT : 1,		CONFIG : 'F U T, 0, 0, 0',
	X =  1102.958  mm,	Y =   975.094  mm,	Z =  1056.986  mm,
	W =    50.535 deg,	P =   -23.426 deg,	R =   -25.981 deg
   GP2:
	UF : 1, UT : 1,
	J1=   180.000 deg,	J2=   150.000 deg
};
P[739]{
   GP1:
	UF : 1, UT : 1,		CONFIG : 'F U T, 0, 0, 0',
	X =   851.887  mm,	Y =   977.237  mm,	Z =  1067.701  mm,
	W =    50.535 deg,	P =   -23.426 deg,	R =   -25.981 deg
   GP2:
	UF : 1, UT : 1,
	J1=   180.000 deg,	J2=   150.000 deg
};
P[740]{
   GP1:
	UF : 1, UT : 1,		CONFIG : 'F U T, 0, 0, 0',
	X =   626.208  mm,	Y =  1096.450  mm,	Z =  1381.774  mm,
	W =    61.728 deg,	P =   -31.893 deg,	R =   -10.883 deg
   GP2:
	UF : 1, UT : 1,
	J1=   180.000 deg,	J2=   150.000 deg
};
P[741]{
   GP1:
	UF : 1, UT : 1,		CONFIG : 'N U T, 0, 0, 0',
	X =   758.466  mm,	Y =  -545.960  mm,	Z =   772.606  mm,
	W =    33.386 deg,	P =   -31.996 deg,	R =   -21.225 deg
   GP2:
	UF : 1, UT : 1,
	J1=   180.000 deg,	J2=  -150.000 deg
};
P[742]{
   GP1:
	UF : 1, UT : 1,		CONFIG : 'N U T, 0, 0, 0',
	X =   710.278  mm,	Y =  -477.960  mm,	Z =   772.606  mm,
	W =    33.386 deg,	P =   -31.996 deg,	R =    -8.428 deg
   GP2:
	UF : 1, UT : 1,
	J1=   180.000 deg,	J2=  -150.000 deg
};
P[743]{
   GP1:
	UF : 1, UT : 1,		CONFIG : 'N U T, 0, 0, 0',
	X =  1905.343  mm,	Y = -1477.017  mm,	Z =  1025.975  mm,
	W =   -39.881 deg,	P =    23.853 deg,	R =    23.904 deg
   GP2:
	UF : 1, UT : 1,
	J1=   180.000 deg,	J2=   -90.000 deg
};
P[744]{
   GP1:
	UF : 1, UT : 1,		CONFIG : 'N U T, 0, 0, 0',
	X =  1932.126  mm,	Y = -1480.053  mm,	Z =  1024.380  mm,
	W =   -43.541 deg,	P =    14.557 deg,	R =    14.831 deg
   GP2:
	UF : 1, UT : 1,
	J1=   180.000 deg,	J2=   -90.000 deg
};
P[745]{
   GP1:
	UF : 1, UT : 1,		CONFIG : 'N U T, 0, 0, 0',
	X =  1967.611  mm,	Y = -1478.561  mm,	Z =  1026.042  mm,
	W =   -43.535 deg,	P =    14.558 deg,	R =    14.822 deg
   GP2:
	UF : 1, UT : 1,
	J1=   180.000 deg,	J2=   -90.000 deg
};
P[746]{
   GP1:
	UF : 1, UT : 1,		CONFIG : 'N U T, 0, 0, 0',
	X =  2000.593  mm,	Y = -1497.735  mm,	Z =  1025.630  mm,
	W =   -43.543 deg,	P =    14.556 deg,	R =   -14.021 deg
   GP2:
	UF : 1, UT : 1,
	J1=   180.000 deg,	J2=   -90.000 deg
};
P[747]{
   GP1:
	UF : 1, UT : 1,		CONFIG : 'N U T, 0, 0, 0',
	X =  2008.768  mm,	Y = -1507.923  mm,	Z =  1025.740  mm,
	W =   -44.808 deg,	P =     8.520 deg,	R =   -27.703 deg
   GP2:
	UF : 1, UT : 1,
	J1=   180.000 deg,	J2=   -90.000 deg
};
P[748]{
   GP1:
	UF : 1, UT : 1,		CONFIG : 'N U T, 0, 0, 0',
	X =  1901.875  mm,	Y =  1465.160  mm,	Z =  1036.238  mm,
	W =    41.263 deg,	P =    19.805 deg,	R =   -17.225 deg
   GP2:
	UF : 1, UT : 1,
	J1=   180.000 deg,	J2=    90.000 deg
};
P[749]{
   GP1:
	UF : 1, UT : 1,		CONFIG : 'N U T, 0, 0, 0',
	X =  1934.116  mm,	Y =  1464.614  mm,	Z =  1037.732  mm,
	W =    41.277 deg,	P =    19.801 deg,	R =   -17.230 deg
   GP2:
	UF : 1, UT : 1,
	J1=   180.000 deg,	J2=    90.000 deg
};
P[750]{
   GP1:
	UF : 1, UT : 1,		CONFIG : 'N U T, 0, 0, 0',
	X =  1965.909  mm,	Y =  1468.963  mm,	Z =  1032.171  mm,
	W =    41.272 deg,	P =    19.803 deg,	R =   -17.223 deg
   GP2:
	UF : 1, UT : 1,
	J1=   180.000 deg,	J2=    90.000 deg
};
P[751]{
   GP1:
	UF : 1, UT : 1,		CONFIG : 'N U T, 0, 0, 0',
	X =  1996.605  mm,	Y =  1480.121  mm,	Z =  1030.618  mm,
	W =    41.277 deg,	P =    19.801 deg,	R =     6.735 deg
   GP2:
	UF : 1, UT : 1,
	J1=   180.000 deg,	J2=    90.000 deg
};
P[752]{
   GP1:
	UF : 1, UT : 1,		CONFIG : 'N U T, 0, 0, 0',
	X =  1999.792  mm,	Y =  1488.994  mm,	Z =  1027.439  mm,
	W =    43.863 deg,	P =    11.272 deg,	R =    16.919 deg
   GP2:
	UF : 1, UT : 1,
	J1=   180.000 deg,	J2=    90.000 deg
};
P[753]{
   GP1:
	UF : 1, UT : 1,		CONFIG : 'N U T, 0, 0, 0',
	X =  1637.861  mm,	Y = -1415.325  mm,	Z =  1029.238  mm,
	W =   -42.847 deg,	P =   -15.300 deg,	R =    39.122 deg
   GP2:
	UF : 1, UT : 1,
	J1=   180.000 deg,	J2=  -125.000 deg
};
P[754]{
   GP1:
	UF : 1, UT : 1,		CONFIG : 'N U T, 0, 0, 0',
	X =  1647.655  mm,	Y = -1408.291  mm,	Z =  1027.027  mm,
	W =   -42.573 deg,	P =   -16.796 deg,	R =    40.474 deg
   GP2:
	UF : 1, UT : 1,
	J1=   180.000 deg,	J2=  -125.000 deg
};
P[755]{
   GP1:
	UF : 1, UT : 1,		CONFIG : 'N U T, 0, 0, 0',
	X =  1660.943  mm,	Y = -1400.277  mm,	Z =  1026.065  mm,
	W =   -42.573 deg,	P =   -16.796 deg,	R =    43.536 deg
   GP2:
	UF : 1, UT : 1,
	J1=   180.000 deg,	J2=  -125.000 deg
};
P[756]{
   GP1:
	UF : 1, UT : 1,		CONFIG : 'N U T, 0, 0, 0',
	X =  1662.852  mm,	Y = -1393.480  mm,	Z =  1032.390  mm,
	W =   -44.235 deg,	P =   -18.485 deg,	R =    48.309 deg
   GP2:
	UF : 1, UT : 1,
	J1=   180.000 deg,	J2=  -125.000 deg
};
P[757]{
   GP1:
	UF : 1, UT : 1,		CONFIG : 'F U T, 0, 0, 0',
	X =  1104.853  mm,	Y =  1006.203  mm,	Z =  1025.639  mm,
	W =    44.130 deg,	P =    -6.203 deg,	R =   -51.549 deg
   GP2:
	UF : 1, UT : 1,
	J1=   180.000 deg,	J2=   150.000 deg
};
P[758]{
   GP1:
	UF : 1, UT : 1,		CONFIG : 'F U T, 0, 0, 0',
	X =  1114.844  mm,	Y =  1000.704  mm,	Z =  1027.080  mm,
	W =    43.014 deg,	P =    -7.268 deg,	R =   -34.946 deg
   GP2:
	UF : 1, UT : 1,
	J1=   180.000 deg,	J2=   150.000 deg
};
P[759]{
   GP1:
	UF : 1, UT : 1,		CONFIG : 'F U T, 0, 0, 0',
	X =  1125.597  mm,	Y =   997.219  mm,	Z =  1027.206  mm,
	W =    42.651 deg,	P =   -14.126 deg,	R =   -20.722 deg
   GP2:
	UF : 1, UT : 1,
	J1=   180.000 deg,	J2=   150.000 deg
};
P[760]{
   GP1:
	UF : 1, UT : 1,		CONFIG : 'F U T, 0, 0, 0',
	X =  1138.321  mm,	Y =   996.177  mm,	Z =  1027.210  mm,
	W =    42.651 deg,	P =   -14.126 deg,	R =   -27.080 deg
   GP2:
	UF : 1, UT : 1,
	J1=   180.000 deg,	J2=   150.000 deg
};
P[761]{
   GP1:
	UF : 1, UT : 1,		CONFIG : 'N U T, 0, 0, 0',
	X =  2788.736  mm,	Y = -1483.274  mm,	Z =   933.541  mm,
	W =   -37.771 deg,	P =   -31.405 deg,	R =    42.828 deg
   GP2:
	UF : 1, UT : 1,
	J1=   100.000 deg,	J2=   -90.000 deg
};
P[762]{
   GP1:
	UF : 1, UT : 1,		CONFIG : 'N U T, 0, 0, 0',
	X =  2790.127  mm,	Y = -1512.097  mm,	Z =   933.343  mm,
	W =   -37.782 deg,	P =   -31.394 deg,	R =    42.842 deg
   GP2:
	UF : 1, UT : 1,
	J1=   100.000 deg,	J2=   -90.000 deg
};
P[763]{
   GP1:
	UF : 1, UT : 1,		CONFIG : 'N U T, 0, 0, 0',
	X =  2777.828  mm,	Y = -1541.019  mm,	Z =   932.405  mm,
	W =   -42.870 deg,	P =   -22.985 deg,	R =    39.985 deg
   GP2:
	UF : 1, UT : 1,
	J1=   100.000 deg,	J2=   -90.000 deg
};
P[764]{
   GP1:
	UF : 1, UT : 1,		CONFIG : 'N U T, 0, 0, 0',
	X =  2762.396  mm,	Y = -1555.396  mm,	Z =   929.477  mm,
	W =   -45.718 deg,	P =   -14.892 deg,	R =    35.274 deg
   GP2:
	UF : 1, UT : 1,
	J1=   100.000 deg,	J2=   -90.000 deg
};
P[765]{
   GP1:
	UF : 1, UT : 1,		CONFIG : 'N U T, 0, 0, 0',
	X =  2731.844  mm,	Y = -1574.335  mm,	Z =   920.084  mm,
	W =   -45.718 deg,	P =   -14.891 deg,	R =    30.406 deg
   GP2:
	UF : 1, UT : 1,
	J1=   100.000 deg,	J2=   -90.000 deg
};
P[766]{
   GP1:
	UF : 1, UT : 1,		CONFIG : 'N U T, 0, 0, 0',
	X =  2725.103  mm,	Y = -1575.819  mm,	Z =   919.847  mm,
	W =   -45.718 deg,	P =   -14.891 deg,	R =    18.309 deg
   GP2:
	UF : 1, UT : 1,
	J1=   100.000 deg,	J2=   -90.000 deg
};
P[767]{
   GP1:
	UF : 1, UT : 1,		CONFIG : 'N U T, 0, 0, 0',
	X =  2712.522  mm,	Y = -1579.347  mm,	Z =   916.110  mm,
	W =   -45.718 deg,	P =   -14.891 deg,	R =     6.077 deg
   GP2:
	UF : 1, UT : 1,
	J1=   100.000 deg,	J2=   -90.000 deg
};
P[768]{
   GP1:
	UF : 1, UT : 1,		CONFIG : 'N U T, 0, 0, 0',
	X =  1082.860  mm,	Y =     -.638  mm,	Z =   529.898  mm,
	W =    48.292 deg,	P =    28.213 deg,	R =    20.411 deg
   GP2:
	UF : 1, UT : 1,
	J1=    80.000 deg,	J2=    90.000 deg
};
P[769]{
   GP1:
	UF : 1, UT : 1,		CONFIG : 'N U T, 0, 0, 0',
	X =  2684.760  mm,	Y = -1581.022  mm,	Z =   910.051  mm,
	W =   -45.718 deg,	P =   -14.891 deg,	R =     6.077 deg
   GP2:
	UF : 1, UT : 1,
	J1=   100.000 deg,	J2=   -90.000 deg
};
P[770]{
   GP1:
	UF : 1, UT : 1,		CONFIG : 'N U T, 0, 0, 0',
	X =  2833.414  mm,	Y =  1483.559  mm,	Z =   885.495  mm,
	W =     1.862 deg,	P =   -42.072 deg,	R =    -2.894 deg
   GP2:
	UF : 1, UT : 1,
	J1=    95.000 deg,	J2=    90.000 deg
};
P[771]{
   GP1:
	UF : 1, UT : 1,		CONFIG : 'N U T, 0, 0, 0',
	X =  2833.081  mm,	Y =  1508.177  mm,	Z =   884.362  mm,
	W =     1.851 deg,	P =   -42.070 deg,	R =    -2.890 deg
   GP2:
	UF : 1, UT : 1,
	J1=    95.000 deg,	J2=    90.000 deg
};
P[772]{
   GP1:
	UF : 1, UT : 1,		CONFIG : 'N U T, 0, 0, 0',
	X =  2826.705  mm,	Y =  1541.371  mm,	Z =   879.685  mm,
	W =    47.457 deg,	P =    -2.512 deg,	R =   -28.093 deg
   GP2:
	UF : 1, UT : 1,
	J1=    95.000 deg,	J2=    90.000 deg
};
P[773]{
   GP1:
	UF : 1, UT : 1,		CONFIG : 'N U T, 0, 0, 0',
	X =  2808.617  mm,	Y =  1556.143  mm,	Z =   878.386  mm,
	W =    47.469 deg,	P =    -2.511 deg,	R =   -28.096 deg
   GP2:
	UF : 1, UT : 1,
	J1=    95.000 deg,	J2=    90.000 deg
};
P[774]{
   GP1:
	UF : 1, UT : 1,		CONFIG : 'N U T, 0, 0, 0',
	X =  2772.622  mm,	Y =  1570.522  mm,	Z =   877.279  mm,
	W =    47.469 deg,	P =    -2.511 deg,	R =   -28.096 deg
   GP2:
	UF : 1, UT : 1,
	J1=    95.000 deg,	J2=    90.000 deg
};
P[775]{
   GP1:
	UF : 1, UT : 1,		CONFIG : 'N U T, 0, 0, 0',
	X =  2766.040  mm,	Y =  1572.698  mm,	Z =   875.804  mm,
	W =    46.964 deg,	P =     8.281 deg,	R =   -26.942 deg
   GP2:
	UF : 1, UT : 1,
	J1=    95.000 deg,	J2=    90.000 deg
};
P[776]{
   GP1:
	UF : 1, UT : 1,		CONFIG : 'N U T, 0, 0, 0',
	X =  2756.734  mm,	Y =  1575.818  mm,	Z =   872.094  mm,
	W =    47.296 deg,	P =    13.421 deg,	R =   -20.078 deg
   GP2:
	UF : 1, UT : 1,
	J1=    94.995 deg,	J2=    90.000 deg
};
P[777]{
   GP1:
	UF : 1, UT : 1,		CONFIG : 'N U T, 0, 0, 0',
	X =  2725.010  mm,	Y =  1574.875  mm,	Z =   871.699  mm,
	W =    46.312 deg,	P =    12.118 deg,	R =   -20.583 deg
   GP2:
	UF : 1, UT : 1,
	J1=    95.000 deg,	J2=    90.000 deg
};
P[778]{
   GP1:
	UF : 1, UT : 1,		CONFIG : 'N U T, 0, 0, 0',
	X =  1684.563  mm,	Y =   458.656  mm,	Z =   830.406  mm,
	W =    39.866 deg,	P =   -22.888 deg,	R =   -65.013 deg
   GP2:
	UF : 1, UT : 1,
	J1=   -90.000 deg,	J2=   -90.000 deg
};
P[779]{
   GP1:
	UF : 1, UT : 1,		CONFIG : 'N U T, 0, 0, 0',
	X =  1685.493  mm,	Y =   473.679  mm,	Z =   828.230  mm,
	W =    39.866 deg,	P =   -22.887 deg,	R =   -65.013 deg
   GP2:
	UF : 1, UT : 1,
	J1=   -90.000 deg,	J2=   -90.000 deg
};
P[780]{
   GP1:
	UF : 1, UT : 1,		CONFIG : 'N U T, 0, 0, 0',
	X =  1685.563  mm,	Y =   480.822  mm,	Z =   829.093  mm,
	W =    39.867 deg,	P =   -22.888 deg,	R =   -69.837 deg
   GP2:
	UF : 1, UT : 1,
	J1=   -90.000 deg,	J2=   -90.000 deg
};
P[781]{
   GP1:
	UF : 1, UT : 1,		CONFIG : 'N U T, 0, 0, 0',
	X =  1687.491  mm,	Y =   484.680  mm,	Z =   827.711  mm,
	W =    39.867 deg,	P =   -22.888 deg,	R =   -70.971 deg
   GP2:
	UF : 1, UT : 1,
	J1=   -90.000 deg,	J2=   -90.000 deg
};
P[782]{
   GP1:
	UF : 1, UT : 1,		CONFIG : 'N U T, 0, 0, 0',
	X =  1708.839  mm,	Y =   554.633  mm,	Z =   827.423  mm,
	W =    39.871 deg,	P =   -22.884 deg,	R =   -70.976 deg
   GP2:
	UF : 1, UT : 1,
	J1=   -90.000 deg,	J2=   -90.000 deg
};
P[783]{
   GP1:
	UF : 1, UT : 1,		CONFIG : 'N U T, 0, 0, 0',
	X =  1711.676  mm,	Y =   557.080  mm,	Z =   826.531  mm,
	W =    39.870 deg,	P =   -22.884 deg,	R =   -74.846 deg
   GP2:
	UF : 1, UT : 1,
	J1=   -90.000 deg,	J2=   -90.000 deg
};
P[784]{
   GP1:
	UF : 1, UT : 1,		CONFIG : 'N U T, 0, 0, 0',
	X =  1712.809  mm,	Y =   560.962  mm,	Z =   826.801  mm,
	W =    39.866 deg,	P =   -22.883 deg,	R =   -82.536 deg
   GP2:
	UF : 1, UT : 1,
	J1=   -90.000 deg,	J2=   -90.000 deg
};
P[785]{
   GP1:
	UF : 1, UT : 1,		CONFIG : 'N U T, 0, 0, 0',
	X =  1845.680  mm,	Y =   825.086  mm,	Z =   832.601  mm,
	W =    14.309 deg,	P =   -43.038 deg,	R =   -40.623 deg
   GP2:
	UF : 1, UT : 1,
	J1=   -89.991 deg,	J2=   -89.999 deg
};
P[786]{
   GP1:
	UF : 1, UT : 1,		CONFIG : 'N U T, 0, 0, 0',
	X =  2547.891  mm,	Y =   822.808  mm,	Z =   -72.485  mm,
	W =   -31.199 deg,	P =     9.620 deg,	R =   105.426 deg
   GP2:
	UF : 1, UT : 1,
	J1=    80.000 deg,	J2=   -90.000 deg
};
P[787]{
   GP1:
	UF : 1, UT : 1,		CONFIG : 'N U T, 0, 0, 0',
	X =  2549.025  mm,	Y =   813.653  mm,	Z =   -72.568  mm,
	W =   -32.484 deg,	P =     1.246 deg,	R =    91.954 deg
   GP2:
	UF : 1, UT : 1,
	J1=    80.000 deg,	J2=   -90.000 deg
};
P[788]{
   GP1:
	UF : 1, UT : 1,		CONFIG : 'N U T, 0, 0, 0',
	X =  2556.443  mm,	Y =   796.316  mm,	Z =   -71.740  mm,
	W =   -29.311 deg,	P =   -14.722 deg,	R =   104.313 deg
   GP2:
	UF : 0, UT : 1,
	J1=    80.000 deg,	J2=   -90.000 deg
};
P[789]{
   GP1:
	UF : 1, UT : 1,		CONFIG : 'N U T, 0, 0, 0',
	X =  2576.844  mm,	Y =   790.013  mm,	Z =   -76.345  mm,
	W =    -3.324 deg,	P =   -34.459 deg,	R =   105.041 deg
   GP2:
	UF : 0, UT : 1,
	J1=    80.000 deg,	J2=   -90.000 deg
};
P[790]{
   GP1:
	UF : 1, UT : 1,		CONFIG : 'N U T, 0, 0, 0',
	X =  2600.397  mm,	Y =   789.960  mm,	Z =   -81.033  mm,
	W =    -3.272 deg,	P =   -34.453 deg,	R =   105.003 deg
   GP2:
	UF : 0, UT : 1,
	J1=    80.000 deg,	J2=   -90.000 deg
};
P[791]{
   GP1:
	UF : 1, UT : 1,		CONFIG : 'N U T, 0, 0, 0',
	X =  2617.219  mm,	Y =   781.118  mm,	Z =   -82.622  mm,
	W =     3.036 deg,	P =   -34.484 deg,	R =    65.941 deg
   GP2:
	UF : 1, UT : 1,
	J1=    80.000 deg,	J2=   -90.000 deg
};
P[792]{
   GP1:
	UF : 1, UT : 1,		CONFIG : 'N U T, 0, 0, 0',
	X =  2627.491  mm,	Y =   762.062  mm,	Z =   -83.870  mm,
	W =   -15.099 deg,	P =   -26.030 deg,	R =    67.737 deg
   GP2:
	UF : 0, UT : 1,
	J1=    80.000 deg,	J2=   -90.000 deg
};
P[793]{
   GP1:
	UF : 1, UT : 1,		CONFIG : 'F U T, 0, 0, 0',
	X =   419.331  mm,	Y =  1026.789  mm,	Z =  1609.020  mm,
	W =    71.318 deg,	P =     7.769 deg,	R =   -20.454 deg
   GP2:
	UF : 1, UT : 1,
	J1=   180.000 deg,	J2=   150.000 deg
};
/END
